// TIA Portal V20 export
// export: Created 2026-04-18T06:33:56.6460483Z, ExportSetting WithDefaults, DisplayName Totally Integrated Automation Portal, DisplayVersion V20, DisplayName TIA Portal Openness, DisplayVersion V20, DisplayName TIA Portal Version Control Interface, DisplayVersion V20, DisplayName STEP 7 Professional, DisplayVersion V20, DisplayName STEP 7 Safety, DisplayVersion V20, DisplayName WinCC Basic/Comfort/Advanced, DisplayVersion V20
TYPE "UDT_ControlValve"
// stored: IsFailsafeCompliant false
   STRUCT
      valveTag : String[16] := 'V-000';
      valveType : Int := 1;   // 1=Ball 2=Butterfly 3=Diaphragm 4=Globe 5=Needle
      travelTime : Time := T#4S;
      positionSetpoint : Real := 0.0;   // %
      deadband : Real := 1.5;   // %
      flowLimits { S7_SetPoint := 'True'} : "UDT_AlarmLimits";
      pressureLimits { S7_SetPoint := 'True'} : "UDT_AlarmLimits";
      comment : String[64] := '';
   END_STRUCT;
END_TYPE
